# EPICS autosave request: srsDS345App/Db/srsDS345_settings.req
$(P)FREQ
$(P)VPP
$(P)VRMS
$(P)WAVEFORM
$(P)DCOFFSET
$(P)PHASE
$(P)ZEROPHASE
$(P)INV
$(P)MOD
$(P)TRIG
$(P)TRIGSRC
$(P)MODTYPE
$(P)BURSTCT
$(P)RATE
